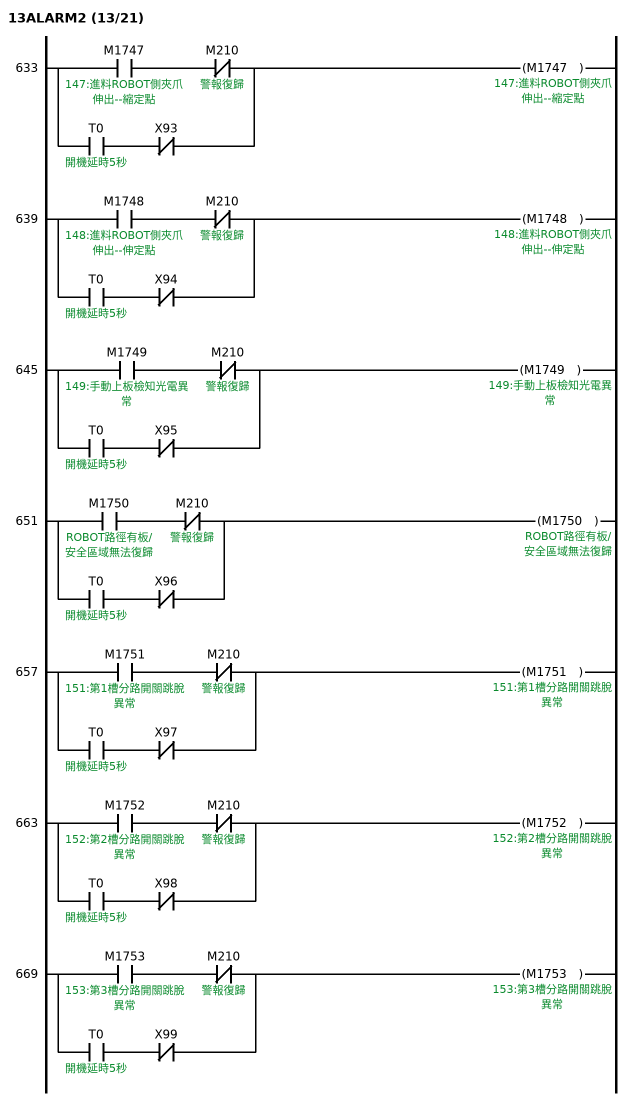
[picture p72: ladder of 13ALARM2, rungs at steps 633 to 669]
633   LD      M1747  ; 147:進料ROBOT側夾爪伸出--縮定點
      ANI     M210  ; 警報復歸
      LD      T0  ; 開機延時5秒
      ANI     X93
      ORB
      OUT     M1747  ; 147:進料ROBOT側夾爪伸出--縮定點
639   LD      M1748  ; 148:進料ROBOT側夾爪伸出--伸定點
      ANI     M210  ; 警報復歸
      LD      T0  ; 開機延時5秒
      ANI     X94
      ORB
      OUT     M1748  ; 148:進料ROBOT側夾爪伸出--伸定點
645   LD      M1749  ; 149:手動上板檢知光電異常
      ANI     M210  ; 警報復歸
      LD      T0  ; 開機延時5秒
      ANI     X95
      ORB
      OUT     M1749  ; 149:手動上板檢知光電異常
651   LD      M1750  ; ROBOT路徑有板/安全區域無法復歸
      ANI     M210  ; 警報復歸
      LD      T0  ; 開機延時5秒
      ANI     X96
      ORB
      OUT     M1750  ; ROBOT路徑有板/安全區域無法復歸
657   LD      M1751  ; 151:第1槽分路開關跳脫異常
      ANI     M210  ; 警報復歸
      LD      T0  ; 開機延時5秒
      ANI     X97
      ORB
      OUT     M1751  ; 151:第1槽分路開關跳脫異常
663   LD      M1752  ; 152:第2槽分路開關跳脫異常
      ANI     M210  ; 警報復歸
      LD      T0  ; 開機延時5秒
      ANI     X98
      ORB
      OUT     M1752  ; 152:第2槽分路開關跳脫異常
669   LD      M1753  ; 153:第3槽分路開關跳脫異常
      ANI     M210  ; 警報復歸
      LD      T0  ; 開機延時5秒
      ANI     X99
      ORB
      OUT     M1753  ; 153:第3槽分路開關跳脫異常
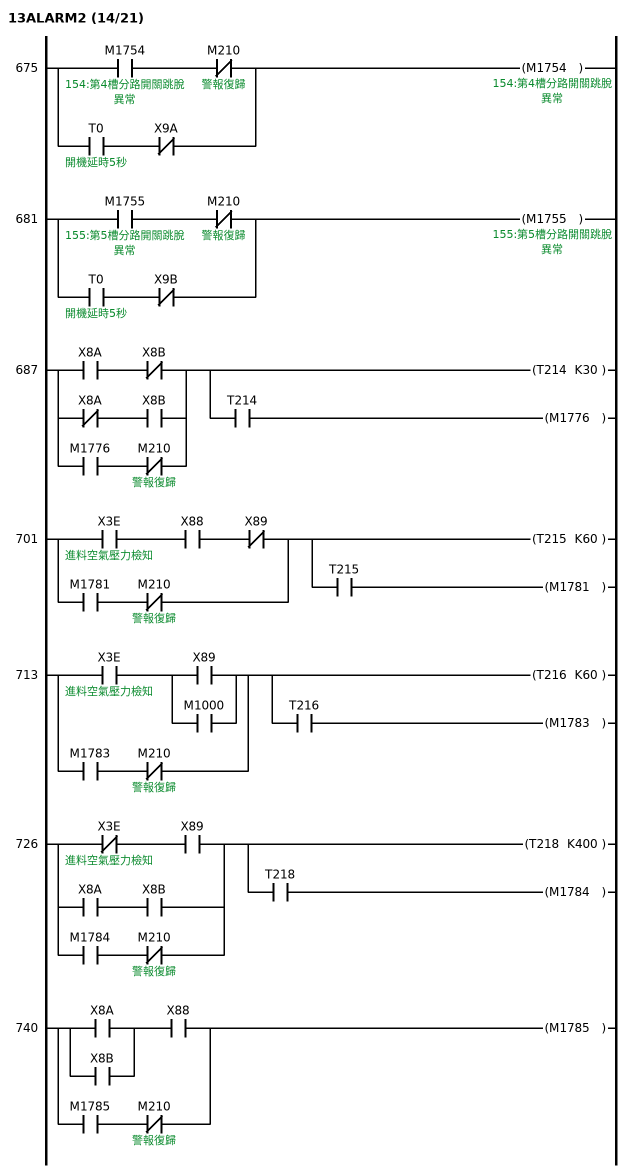
675   LD      M1754  ; 154:第4槽分路開關跳脫異常
      ANI     M210  ; 警報復歸
      LD      T0  ; 開機延時5秒
      ANI     X9A
      ORB
      OUT     M1754  ; 154:第4槽分路開關跳脫異常
681   LD      M1755  ; 155:第5槽分路開關跳脫異常
      ANI     M210  ; 警報復歸
      LD      T0  ; 開機延時5秒
      ANI     X9B
      ORB
      OUT     M1755  ; 155:第5槽分路開關跳脫異常
687   LD      X8A
      ANI     X8B
      LDI     X8A
      AND     X8B
      ORB
      LD      M1776
      ANI     M210  ; 警報復歸
      ORB
      OUT     T214 K30
      AND     T214
      OUT     M1776
701   LD      X3E  ; 進料空氣壓力檢知
      AND     X88
      ANI     X89
      LD      M1781
      ANI     M210  ; 警報復歸
      ORB
      OUT     T215 K60
      AND     T215
      OUT     M1781
713   LD      X3E  ; 進料空氣壓力檢知
      LD      X89
      OR      M1000
      ANB
      LD      M1783
      ANI     M210  ; 警報復歸
      ORB
      OUT     T216 K60
      AND     T216
      OUT     M1783
726   LDI     X3E  ; 進料空氣壓力檢知
      AND     X89
      LD      X8A
      AND     X8B
      ORB
      LD      M1784
      ANI     M210  ; 警報復歸
      ORB
      OUT     T218 K400
      AND     T218
      OUT     M1784
740   LD      X8A
      OR      X8B
      AND     X88
      LD      M1785
      ANI     M210  ; 警報復歸
      ORB
      OUT     M1785
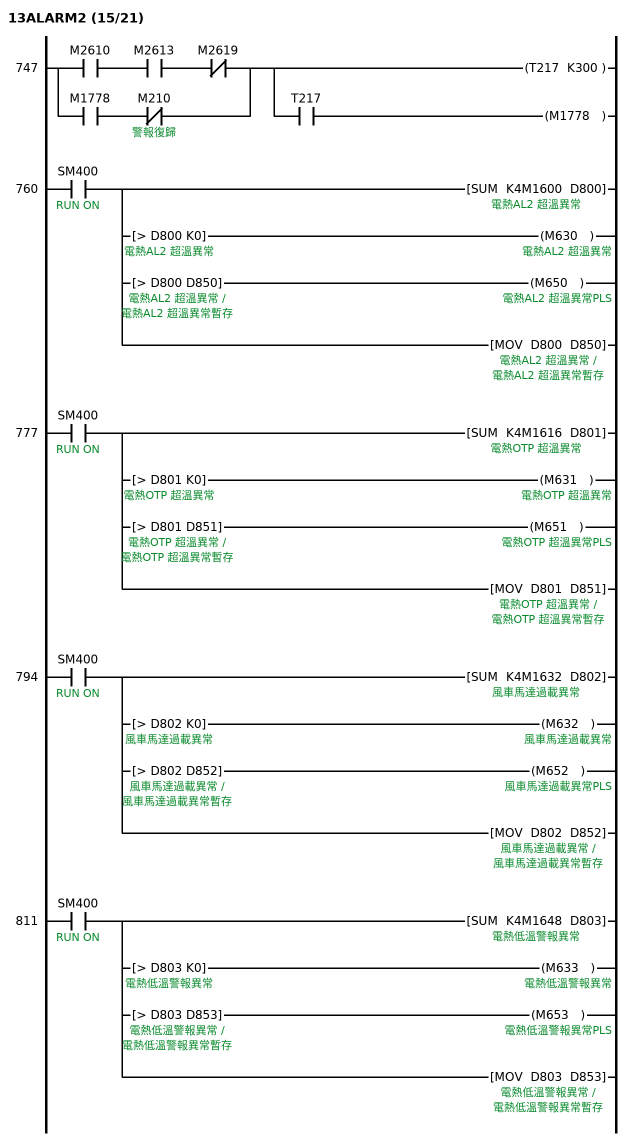
747   LD      M2610
      AND     M2613
      ANI     M2619
      LD      M1778
      ANI     M210  ; 警報復歸
      ORB
      OUT     T217 K300
      AND     T217
      OUT     M1778
760   LD      SM400  ; RUN ON
      SUM     K4M1600 D800  ; #01 電熱AL2 超溫 / 電熱AL2 超溫異常
      MPS
      AND>    D800 K0  ; 電熱AL2 超溫異常
      OUT     M630  ; 電熱AL2 超溫異常
      MRD
      AND>    D800 D850  ; 電熱AL2 超溫異常 / 電熱AL2 超溫異常暫存
      OUT     M650  ; 電熱AL2 超溫異常PLS
      MPP
      MOV     D800 D850
777   LD      SM400  ; RUN ON
      SUM     K4M1616 D801  ; #01 電熱OTP 超溫 / 電熱OTP 超溫異常
      MPS
      AND>    D801 K0  ; 電熱OTP 超溫異常
      OUT     M631  ; 電熱OTP 超溫異常
      MRD
      AND>    D801 D851  ; 電熱OTP 超溫異常 / 電熱OTP 超溫異常暫存
      OUT     M651  ; 電熱OTP 超溫異常PLS
      MPP
      MOV     D801 D851
794   LD      SM400  ; RUN ON
      SUM     K4M1632 D802  ; #01 風車過載 / 風車馬達過載異常
      MPS
      AND>    D802 K0  ; 風車馬達過載異常
      OUT     M632  ; 風車馬達過載異常
      MRD
      AND>    D802 D852  ; 風車馬達過載異常 / 風車馬達過載異常暫存
      OUT     M652  ; 風車馬達過載異常PLS
      MPP
      MOV     D802 D852
811   LD      SM400  ; RUN ON
      SUM     K4M1648 D803  ; #01 低溫警報 / 電熱低溫警報異常
      MPS
      AND>    D803 K0  ; 電熱低溫警報異常
      OUT     M633  ; 電熱低溫警報異常
      MRD
      AND>    D803 D853  ; 電熱低溫警報異常 / 電熱低溫警報異常暫存
      OUT     M653  ; 電熱低溫警報異常PLS
      MPP
      MOV     D803 D853
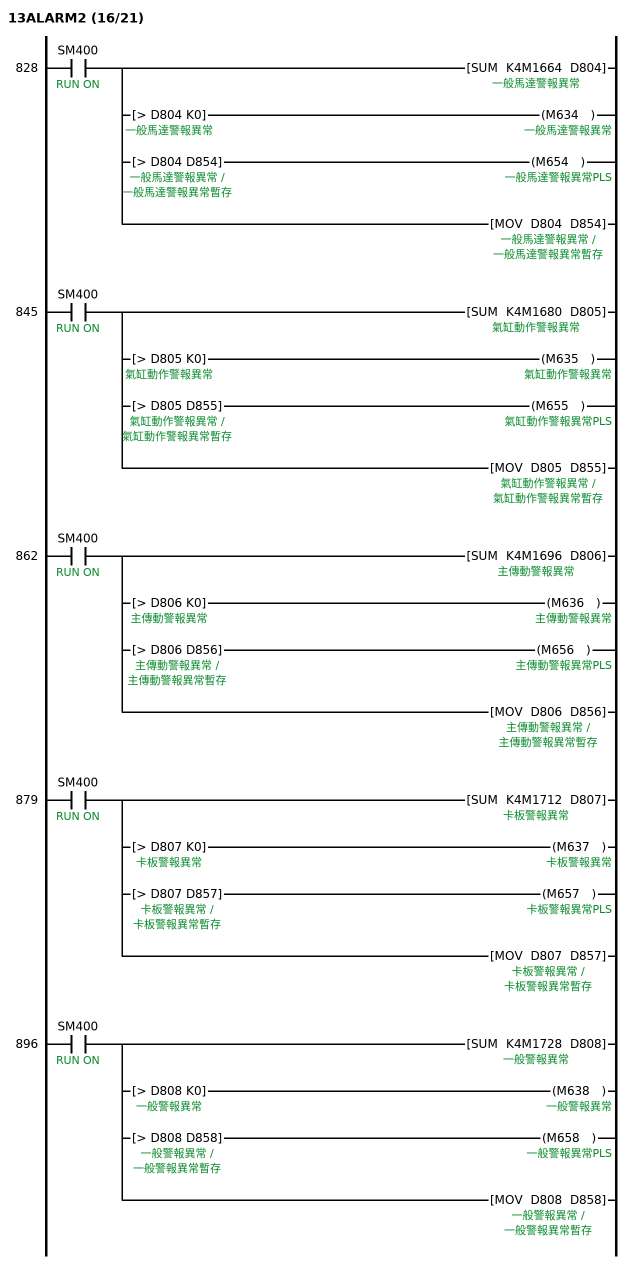
828   LD      SM400  ; RUN ON
      SUM     K4M1664 D804  ; 一般馬達警報異常
      MPS
      AND>    D804 K0  ; 一般馬達警報異常
      OUT     M634  ; 一般馬達警報異常
      MRD
      AND>    D804 D854  ; 一般馬達警報異常 / 一般馬達警報異常暫存
      OUT     M654  ; 一般馬達警報異常PLS
      MPP
      MOV     D804 D854
845   LD      SM400  ; RUN ON
      SUM     K4M1680 D805  ; 氣缸動作警報異常
      MPS
      AND>    D805 K0  ; 氣缸動作警報異常
      OUT     M635  ; 氣缸動作警報異常
      MRD
      AND>    D805 D855  ; 氣缸動作警報異常 / 氣缸動作警報異常暫存
      OUT     M655  ; 氣缸動作警報異常PLS
      MPP
      MOV     D805 D855
862   LD      SM400  ; RUN ON
      SUM     K4M1696 D806  ; 主傳動警報異常
      MPS
      AND>    D806 K0  ; 主傳動警報異常
      OUT     M636  ; 主傳動警報異常
      MRD
      AND>    D806 D856  ; 主傳動警報異常 / 主傳動警報異常暫存
      OUT     M656  ; 主傳動警報異常PLS
      MPP
      MOV     D806 D856
879   LD      SM400  ; RUN ON
      SUM     K4M1712 D807  ; 卡板警報異常
      MPS
      AND>    D807 K0  ; 卡板警報異常
      OUT     M637  ; 卡板警報異常
      MRD
      AND>    D807 D857  ; 卡板警報異常 / 卡板警報異常暫存
      OUT     M657  ; 卡板警報異常PLS
      MPP
      MOV     D807 D857
896   LD      SM400  ; RUN ON
      SUM     K4M1728 D808  ; 一般警報異常
      MPS
      AND>    D808 K0  ; 一般警報異常
      OUT     M638  ; 一般警報異常
      MRD
      AND>    D808 D858  ; 一般警報異常 / 一般警報異常暫存
      OUT     M658  ; 一般警報異常PLS
      MPP
      MOV     D808 D858
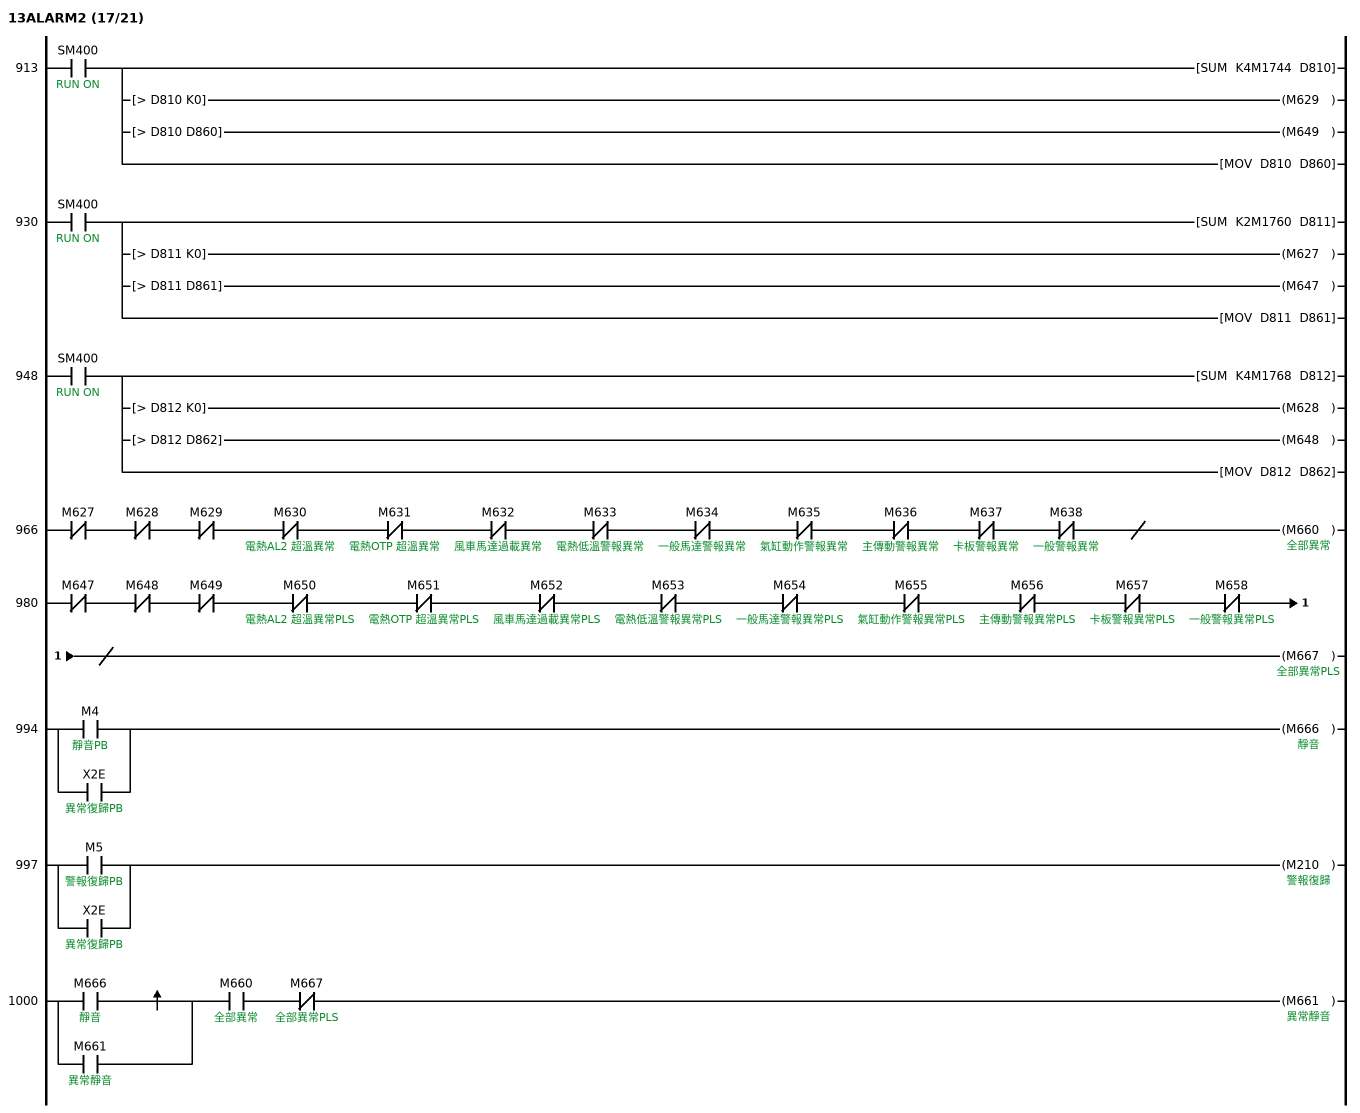
913   LD      SM400  ; RUN ON
      SUM     K4M1744 D810
      MPS
      AND>    D810 K0
      OUT     M629
      MRD
      AND>    D810 D860
      OUT     M649
      MPP
      MOV     D810 D860
930   LD      SM400  ; RUN ON
      SUM     K2M1760 D811
      MPS
      AND>    D811 K0
      OUT     M627
      MRD
      AND>    D811 D861
      OUT     M647
      MPP
      MOV     D811 D861
948   LD      SM400  ; RUN ON
      SUM     K4M1768 D812
      MPS
      AND>    D812 K0
      OUT     M628
      MRD
      AND>    D812 D862
      OUT     M648
      MPP
      MOV     D812 D862
966   LDI     M627
      ANI     M628
      ANI     M629
      ANI     M630  ; 電熱AL2 超溫異常
      ANI     M631  ; 電熱OTP 超溫異常
      ANI     M632  ; 風車馬達過載異常
      ANI     M633  ; 電熱低溫警報異常
      ANI     M634  ; 一般馬達警報異常
      ANI     M635  ; 氣缸動作警報異常
      ANI     M636  ; 主傳動警報異常
      ANI     M637  ; 卡板警報異常
      ANI     M638  ; 一般警報異常
      INV
      OUT     M660  ; 全部異常
980   LDI     M647
      ANI     M648
      ANI     M649
      ANI     M650  ; 電熱AL2 超溫異常PLS
      ANI     M651  ; 電熱OTP 超溫異常PLS
      ANI     M652  ; 風車馬達過載異常PLS
      ANI     M653  ; 電熱低溫警報異常PLS
      ANI     M654  ; 一般馬達警報異常PLS
      ANI     M655  ; 氣缸動作警報異常PLS
      ANI     M656  ; 主傳動警報異常PLS
      ANI     M657  ; 卡板警報異常PLS
      ANI     M658  ; 一般警報異常PLS
      INV
      OUT     M667  ; 全部異常PLS
994   LD      M4  ; 靜音PB
      OR      X2E  ; 異常復歸PB
      OUT     M666  ; 靜音
997   LD      M5  ; 警報復歸PB
      OR      X2E  ; 異常復歸PB
      OUT     M210  ; 警報復歸
1000  LD      M666  ; 靜音
      MEP
      OR      M661  ; 異常靜音
      AND     M660  ; 全部異常
      ANI     M667  ; 全部異常PLS
      OUT     M661  ; 異常靜音
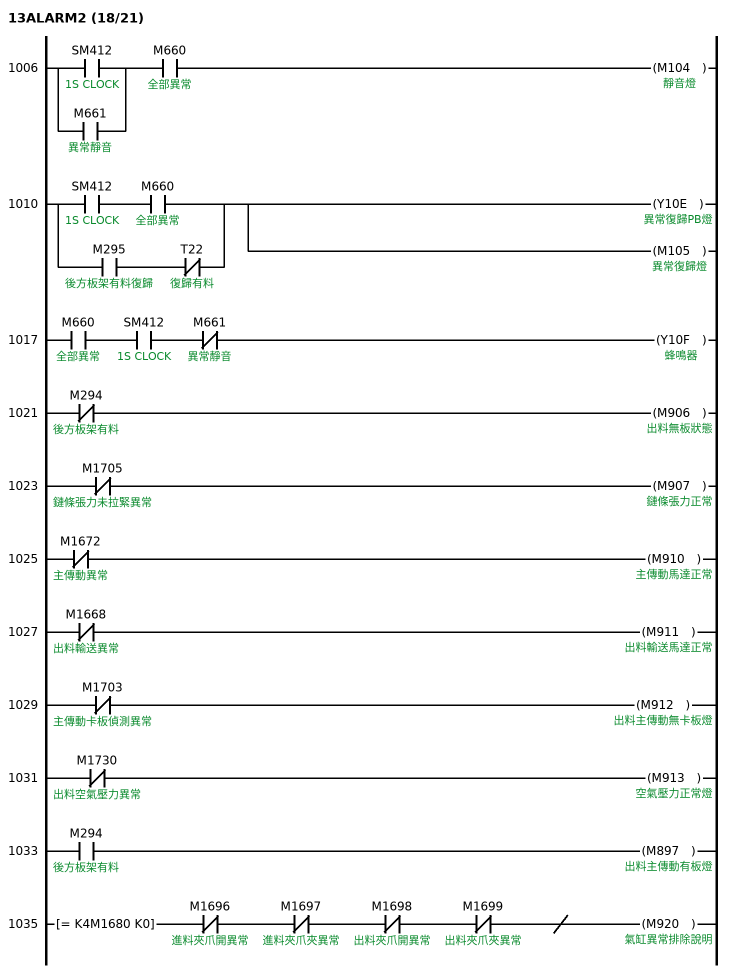
1006  LD      SM412  ; 1S CLOCK
      OR      M661  ; 異常靜音
      AND     M660  ; 全部異常
      OUT     M104  ; 靜音燈
1010  LD      SM412  ; 1S CLOCK
      AND     M660  ; 全部異常
      LD      M295  ; 後方板架有料復歸
      ANI     T22  ; 復歸有料
      ORB
      OUT     Y10E  ; 異常復歸PB燈
      OUT     M105  ; 異常復歸燈
1017  LD      M660  ; 全部異常
      AND     SM412  ; 1S CLOCK
      ANI     M661  ; 異常靜音
      OUT     Y10F  ; 蜂鳴器
1021  LDI     M294  ; 後方板架有料
      OUT     M906  ; 出料無板狀態
1023  LDI     M1705  ; 鏈條張力未拉緊異常
      OUT     M907  ; 鏈條張力正常
1025  LDI     M1672  ; 主傳動異常
      OUT     M910  ; 主傳動馬達正常
1027  LDI     M1668  ; 出料輸送異常
      OUT     M911  ; 出料輸送馬達正常
1029  LDI     M1703  ; 主傳動卡板偵測異常
      OUT     M912  ; 出料主傳動無卡板燈
1031  LDI     M1730  ; 出料空氣壓力異常
      OUT     M913  ; 空氣壓力正常燈
1033  LD      M294  ; 後方板架有料
      OUT     M897  ; 出料主傳動有板燈
1035  LD=     K4M1680 K0  ; 上料手臂前夾爪放異常
      ANI     M1696  ; 進料夾爪開異常
      ANI     M1697  ; 進料夾爪夾異常
      ANI     M1698  ; 出料夾爪開異常
      ANI     M1699  ; 出料夾爪夾異常
      INV
      OUT     M920  ; 氣缸異常排除說明
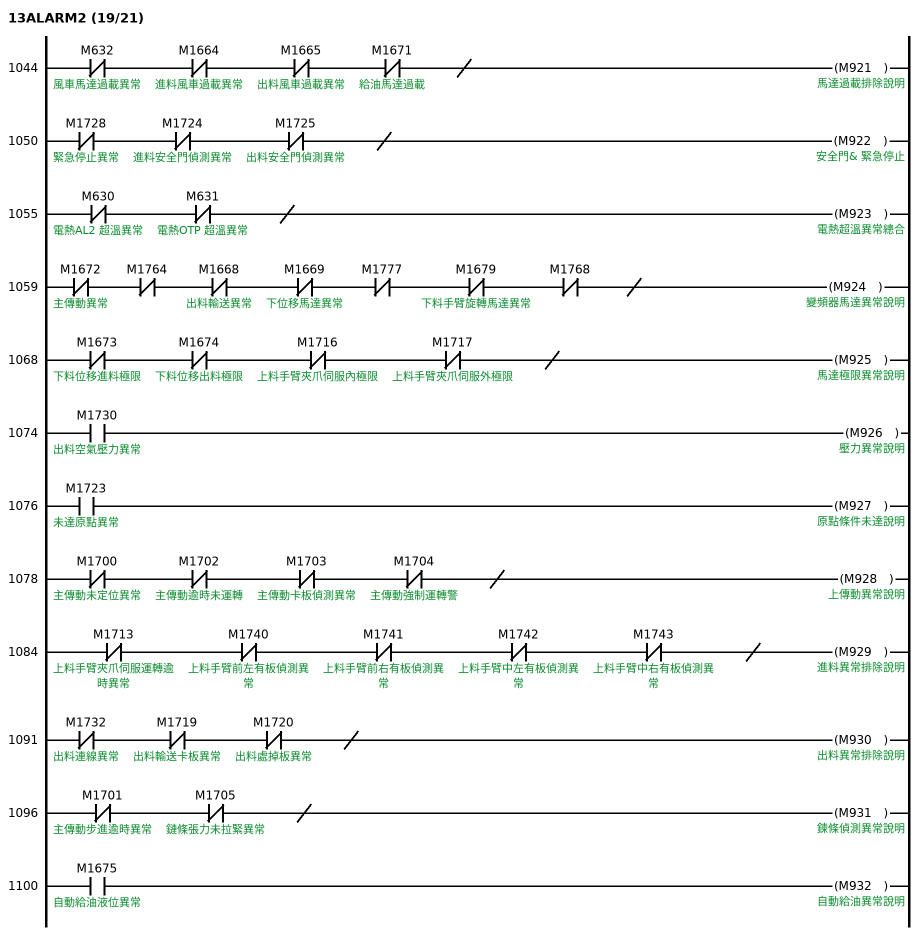
1044  LDI     M632  ; 風車馬達過載異常
      ANI     M1664  ; 進料風車過載異常
      ANI     M1665  ; 出料風車過載異常
      ANI     M1671  ; 給油馬達過載
      INV
      OUT     M921  ; 馬達過載排除說明
1050  LDI     M1728  ; 緊急停止異常
      ANI     M1724  ; 進料安全門偵測異常
      ANI     M1725  ; 出料安全門偵測異常
      INV
      OUT     M922  ; 安全門& 緊急停止
1055  LDI     M630  ; 電熱AL2 超溫異常
      ANI     M631  ; 電熱OTP 超溫異常
      INV
      OUT     M923  ; 電熱超溫異常總合
1059  LDI     M1672  ; 主傳動異常
      ANI     M1764
      ANI     M1668  ; 出料輸送異常
      ANI     M1669  ; 下位移馬達異常
      ANI     M1777
      ANI     M1679  ; 下料手臂旋轉馬達異常
      ANI     M1768
      INV
      OUT     M924  ; 變頻器馬達異常說明
1068  LDI     M1673  ; 下料位移進料極限
      ANI     M1674  ; 下料位移出料極限
      ANI     M1716  ; 上料手臂夾爪伺服內極限
      ANI     M1717  ; 上料手臂夾爪伺服外極限
      INV
      OUT     M925  ; 馬達極限異常說明
1074  LD      M1730  ; 出料空氣壓力異常
      OUT     M926  ; 壓力異常說明
1076  LD      M1723  ; 未達原點異常
      OUT     M927  ; 原點條件未達說明
1078  LDI     M1700  ; 主傳動未定位異常
      ANI     M1702  ; 主傳動逾時未運轉
      ANI     M1703  ; 主傳動卡板偵測異常
      ANI     M1704  ; 主傳動強制運轉警
      INV
      OUT     M928  ; 上傳動異常說明
1084  LDI     M1713  ; 上料手臂夾爪伺服運轉逾時異常
      ANI     M1740  ; 上料手臂前左有板偵測異常
      ANI     M1741  ; 上料手臂前右有板偵測異常
      ANI     M1742  ; 上料手臂中左有板偵測異常
      ANI     M1743  ; 上料手臂中右有板偵測異常
      INV
      OUT     M929  ; 進料異常排除說明
1091  LDI     M1732  ; 出料連線異常
      ANI     M1719  ; 出料輸送卡板異常
      ANI     M1720  ; 出料處掉板異常
      INV
      OUT     M930  ; 出料異常排除說明
1096  LDI     M1701  ; 主傳動步進逾時異常
      ANI     M1705  ; 鏈條張力未拉緊異常
      INV
      OUT     M931  ; 鍊條偵測異常說明
1100  LD      M1675  ; 自動給油液位異常
      OUT     M932  ; 自動給油異常說明
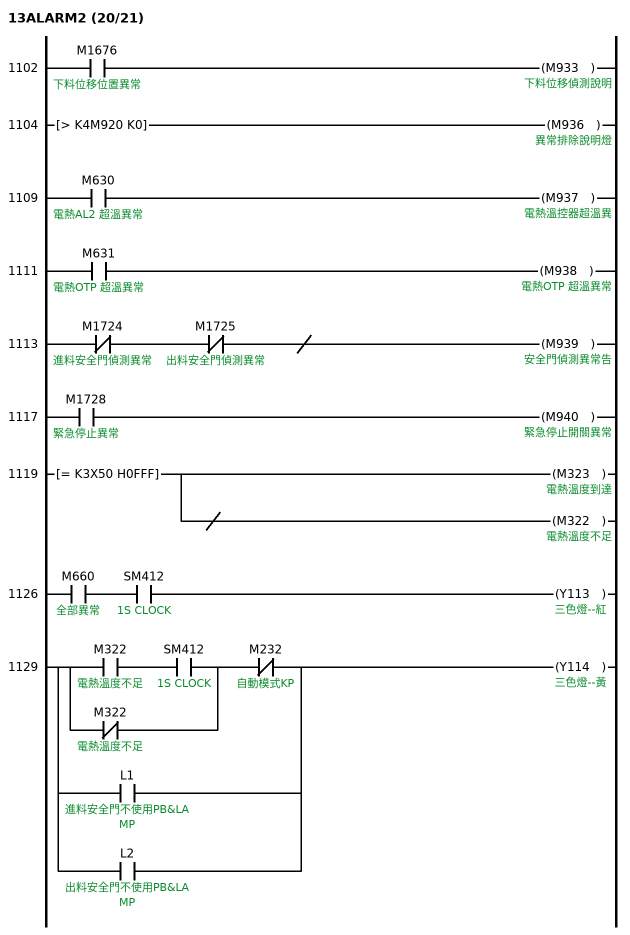
1102  LD      M1676  ; 下料位移位置異常
      OUT     M933  ; 下料位移偵測說明
1104  LD>     K4M920 K0  ; 氣缸異常排除說明
      OUT     M936  ; 異常排除說明燈
1109  LD      M630  ; 電熱AL2 超溫異常
      OUT     M937  ; 電熱溫控器超溫異
1111  LD      M631  ; 電熱OTP 超溫異常
      OUT     M938  ; 電熱OTP 超溫異常
1113  LDI     M1724  ; 進料安全門偵測異常
      ANI     M1725  ; 出料安全門偵測異常
      INV
      OUT     M939  ; 安全門偵測異常告
1117  LD      M1728  ; 緊急停止異常
      OUT     M940  ; 緊急停止開關異常
1119  LD=     K3X50 H0FFF  ; #01 溫度到達AL1
      OUT     M323  ; 電熱溫度到達
      INV
      OUT     M322  ; 電熱溫度不足
1126  LD      M660  ; 全部異常
      AND     SM412  ; 1S CLOCK
      OUT     Y113  ; 三色燈--紅
1129  LD      M322  ; 電熱溫度不足
      AND     SM412  ; 1S CLOCK
      ORI     M322  ; 電熱溫度不足
      ANI     M232  ; 自動模式KP
      OR      L1  ; 進料安全門不使用PB&LAMP
      OR      L2  ; 出料安全門不使用PB&LAMP
      OUT     Y114  ; 三色燈--黃
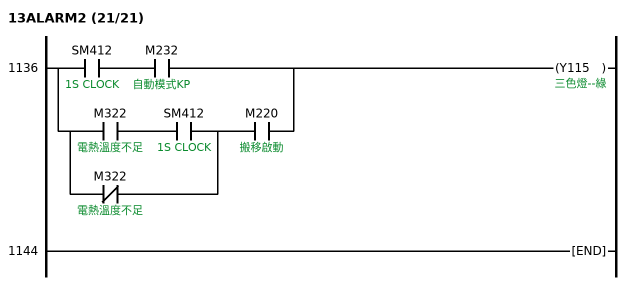
1136  LD      SM412  ; 1S CLOCK
      AND     M232  ; 自動模式KP
      LD      M322  ; 電熱溫度不足
      AND     SM412  ; 1S CLOCK
      ORI     M322  ; 電熱溫度不足
      AND     M220  ; 搬移啟動
      ORB
      OUT     Y115  ; 三色燈--綠
1144  END
END_PROGRAM

PROGRAM 14TIME
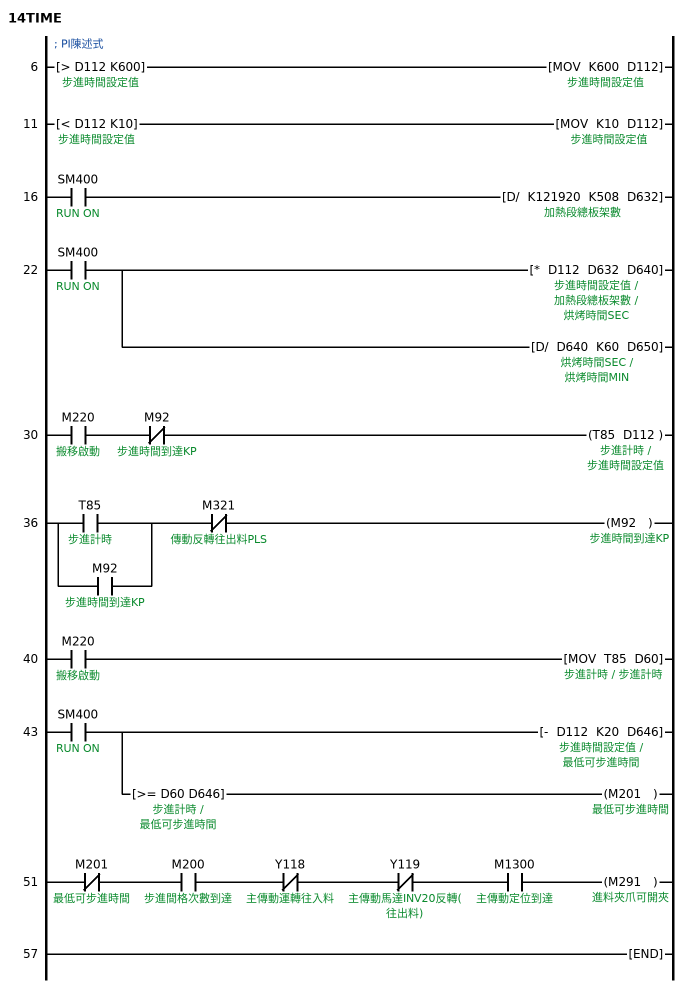
; PI陳述式
6     LD>     D112 K600  ; 步進時間設定值
      MOV     K600 D112
11    LD<     D112 K10  ; 步進時間設定值
      MOV     K10 D112
16    LD      SM400  ; RUN ON
      D/      K121920 K508 D632  ; 加熱段總板架數
22    LD      SM400  ; RUN ON
      *       D112 D632 D640  ; 烘烤時間SEC
      D/      D640 K60 D650  ; 烘烤時間MIN
30    LD      M220  ; 搬移啟動
      ANI     M92  ; 步進時間到達KP
      OUT     T85 D112  ; 步進計時 / 步進時間設定值
36    LD      T85  ; 步進計時
      OR      M92  ; 步進時間到達KP
      ANI     M321  ; 傳動反轉往出料PLS
      OUT     M92  ; 步進時間到達KP
40    LD      M220  ; 搬移啟動
      MOV     T85 D60  ; 步進計時
43    LD      SM400  ; RUN ON
      -       D112 K20 D646  ; 最低可步進時間
      AND>=   D60 D646  ; 步進計時 / 最低可步進時間
      OUT     M201  ; 最低可步進時間
51    LDI     M201  ; 最低可步進時間
      AND     M200  ; 步進間格次數到達
      ANI     Y118  ; 主傳動運轉往入料
      ANI     Y119  ; 主傳動馬達INV20反轉(往出料)
      AND     M1300  ; 主傳動定位到達
      OUT     M291  ; 進料夾爪可開夾
57    END
END_PROGRAM

PROGRAM 15STATUS
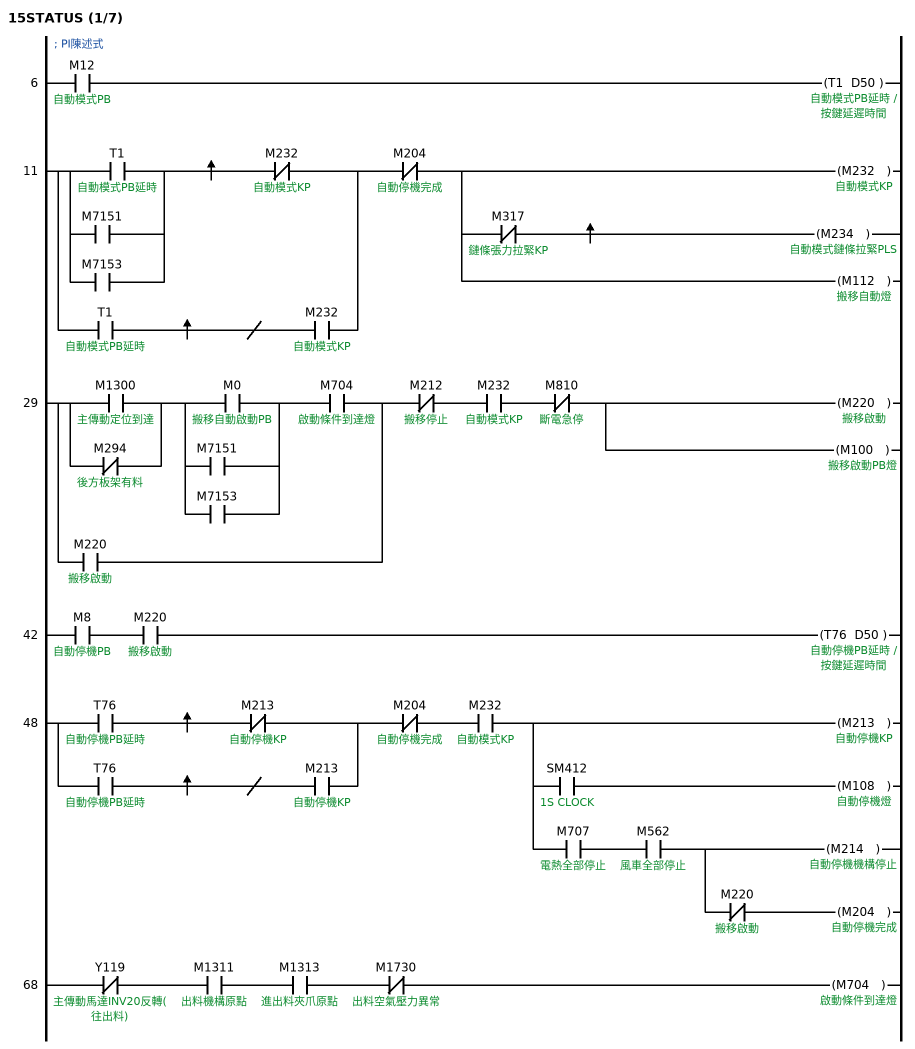
; PI陳述式
6     LD      M12  ; 自動模式PB
      OUT     T1 D50  ; 自動模式PB延時 / 按鍵延遲時間
11    LD      T1  ; 自動模式PB延時
      OR      M7151
      OR      M7153
      MEP
      ANI     M232  ; 自動模式KP
      LD      T1  ; 自動模式PB延時
      MEP
      INV
      AND     M232  ; 自動模式KP
      ORB
      ANI     M204  ; 自動停機完成
      OUT     M232  ; 自動模式KP
      MPS
      ANI     M317  ; 鏈條張力拉緊KP
      MEP
      OUT     M234  ; 自動模式鏈條拉緊PLS
      MPP
      OUT     M112  ; 搬移自動燈
29    LD      M1300  ; 主傳動定位到達
      ORI     M294  ; 後方板架有料
      LD      M0  ; 搬移自動啟動PB
      OR      M7151
      OR      M7153
      ANB
      AND     M704  ; 啟動條件到達燈
      OR      M220  ; 搬移啟動
      ANI     M212  ; 搬移停止
      AND     M232  ; 自動模式KP
      ANI     M810  ; 斷電急停
      OUT     M220  ; 搬移啟動
      OUT     M100  ; 搬移啟動PB燈
42    LD      M8  ; 自動停機PB
      AND     M220  ; 搬移啟動
      OUT     T76 D50  ; 自動停機PB延時 / 按鍵延遲時間
48    LD      T76  ; 自動停機PB延時
      MEP
      ANI     M213  ; 自動停機KP
      LD      T76  ; 自動停機PB延時
      MEP
      INV
      AND     M213  ; 自動停機KP
      ORB
      ANI     M204  ; 自動停機完成
      AND     M232  ; 自動模式KP
      OUT     M213  ; 自動停機KP
      MPS
      AND     SM412  ; 1S CLOCK
      OUT     M108  ; 自動停機燈
      MPP
      AND     M707  ; 電熱全部停止
      AND     M562  ; 風車全部停止
      OUT     M214  ; 自動停機機構停止
      ANI     M220  ; 搬移啟動
      OUT     M204  ; 自動停機完成
68    LDI     Y119  ; 主傳動馬達INV20反轉(往出料)
      AND     M1311  ; 出料機構原點
      AND     M1313  ; 進出料夾爪原點
      ANI     M1730  ; 出料空氣壓力異常
      OUT     M704  ; 啟動條件到達燈
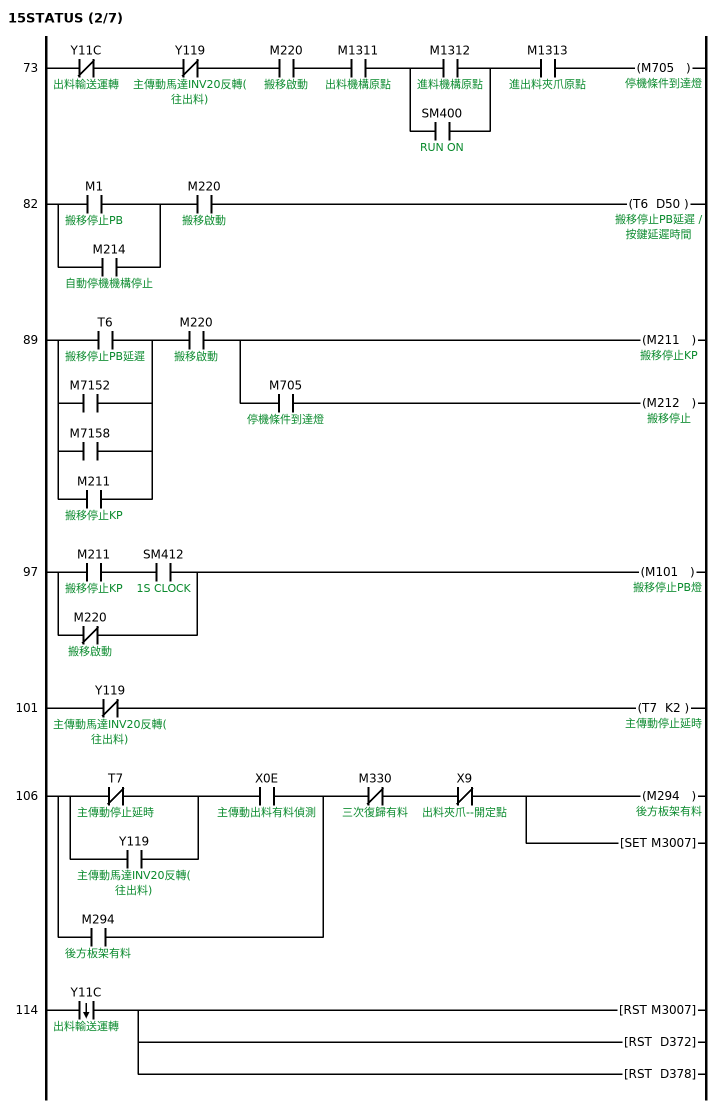
73    LDI     Y11C  ; 出料輸送運轉
      ANI     Y119  ; 主傳動馬達INV20反轉(往出料)
      AND     M220  ; 搬移啟動
      AND     M1311  ; 出料機構原點
      LD      M1312  ; 進料機構原點
      OR      SM400  ; RUN ON
      ANB
      AND     M1313  ; 進出料夾爪原點
      OUT     M705  ; 停機條件到達燈
82    LD      M1  ; 搬移停止PB
      OR      M214  ; 自動停機機構停止
      AND     M220  ; 搬移啟動
      OUT     T6 D50  ; 搬移停止PB延遲 / 按鍵延遲時間
89    LD      T6  ; 搬移停止PB延遲
      OR      M7152
      OR      M7158
      OR      M211  ; 搬移停止KP
      AND     M220  ; 搬移啟動
      OUT     M211  ; 搬移停止KP
      AND     M705  ; 停機條件到達燈
      OUT     M212  ; 搬移停止
97    LD      M211  ; 搬移停止KP
      AND     SM412  ; 1S CLOCK
      ORI     M220  ; 搬移啟動
      OUT     M101  ; 搬移停止PB燈
101   LDI     Y119  ; 主傳動馬達INV20反轉(往出料)
      OUT     T7 K2  ; 主傳動停止延時
106   LDI     T7  ; 主傳動停止延時
      OR      Y119  ; 主傳動馬達INV20反轉(往出料)
      AND     X0E  ; 主傳動出料有料偵測
      OR      M294  ; 後方板架有料
      ANI     M330  ; 三次復歸有料
      ANI     X9  ; 出料夾爪--開定點
      OUT     M294  ; 後方板架有料
      SET     M3007
114   LDF     Y11C  ; 出料輸送運轉
      RST     M3007
      RST     D372
      RST     D378
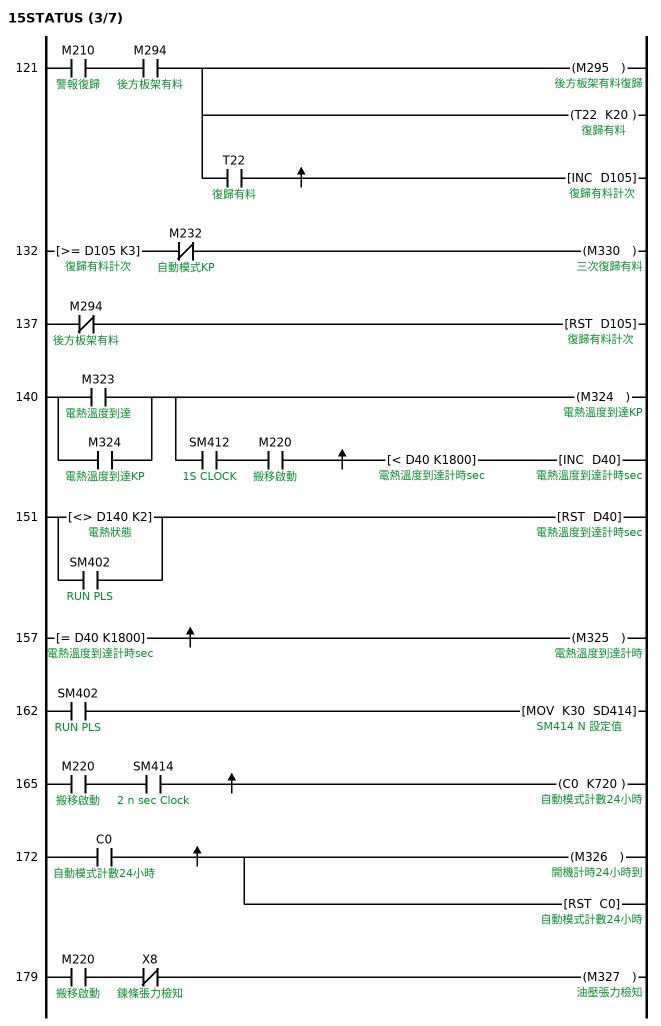
121   LD      M210  ; 警報復歸
      AND     M294  ; 後方板架有料
      OUT     M295  ; 後方板架有料復歸
      OUT     T22 K20  ; 復歸有料
      AND     T22  ; 復歸有料
      MEP
      INC     D105  ; 復歸有料計次
132   LD>=    D105 K3  ; 復歸有料計次
      ANI     M232  ; 自動模式KP
      OUT     M330  ; 三次復歸有料
137   LDI     M294  ; 後方板架有料
      RST     D105  ; 復歸有料計次
140   LD      M323  ; 電熱溫度到達
      OR      M324  ; 電熱溫度到達KP
      OUT     M324  ; 電熱溫度到達KP
      AND     SM412  ; 1S CLOCK
      AND     M220  ; 搬移啟動
      MEP
      AND<    D40 K1800  ; 電熱溫度到達計時sec
      INC     D40
151   LD<>    D140 K2  ; 電熱狀態
      OR      SM402  ; RUN PLS
      RST     D40  ; 電熱溫度到達計時sec
157   LD=     D40 K1800  ; 電熱溫度到達計時sec
      MEP
      OUT     M325  ; 電熱溫度到達計時
162   LD      SM402  ; RUN PLS
      MOV     K30 SD414  ; SM414 N 設定值
165   LD      M220  ; 搬移啟動
      AND     SM414  ; 2 n sec Clock
      MEP
      OUT     C0 K720  ; 自動模式計數24小時
172   LD      C0  ; 自動模式計數24小時
      MEP
      OUT     M326  ; 開機計時24小時到
      RST     C0  ; 自動模式計數24小時
179   LD      M220  ; 搬移啟動
      ANI     X8  ; 鍊條張力檢知
      OUT     M327  ; 油壓張力檢知
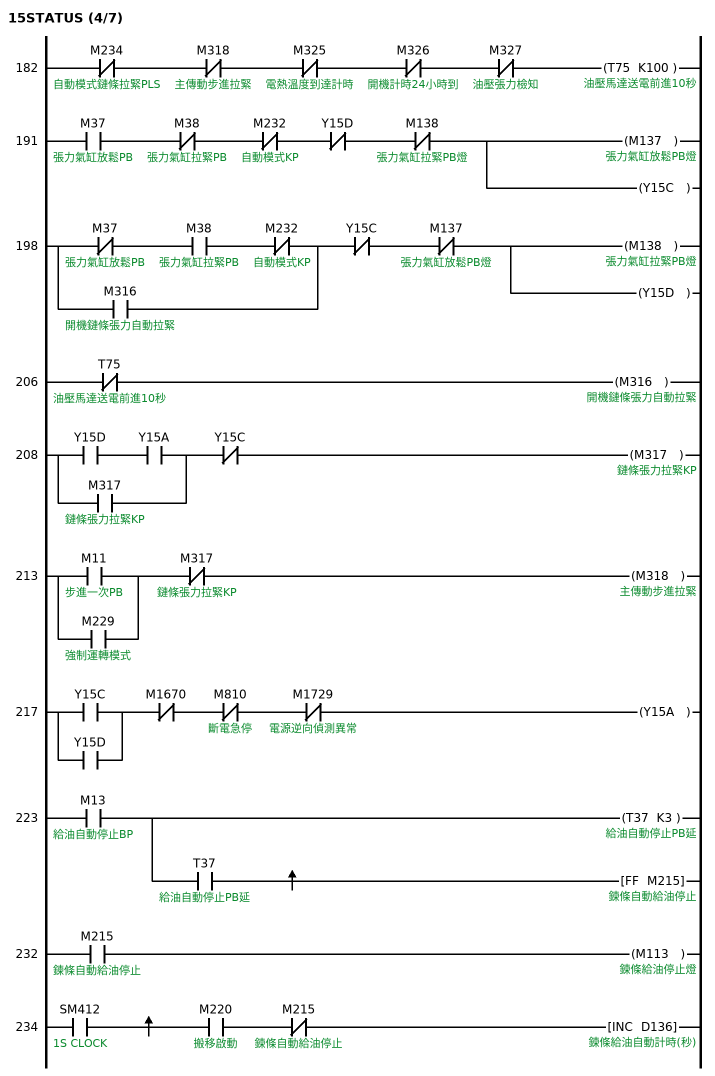
182   LDI     M234  ; 自動模式鏈條拉緊PLS
      ANI     M318  ; 主傳動步進拉緊
      ANI     M325  ; 電熱溫度到達計時
      ANI     M326  ; 開機計時24小時到
      ANI     M327  ; 油壓張力檢知
      OUT     T75 K100  ; 油壓馬達送電前進10秒
191   LD      M37  ; 張力氣缸放鬆PB
      ANI     M38  ; 張力氣缸拉緊PB
      ANI     M232  ; 自動模式KP
      ANI     Y15D
      ANI     M138  ; 張力氣缸拉緊PB燈
      OUT     M137  ; 張力氣缸放鬆PB燈
      OUT     Y15C
198   LDI     M37  ; 張力氣缸放鬆PB
      AND     M38  ; 張力氣缸拉緊PB
      ANI     M232  ; 自動模式KP
      OR      M316  ; 開機鏈條張力自動拉緊
      ANI     Y15C
      ANI     M137  ; 張力氣缸放鬆PB燈
      OUT     M138  ; 張力氣缸拉緊PB燈
      OUT     Y15D
206   LDI     T75  ; 油壓馬達送電前進10秒
      OUT     M316  ; 開機鏈條張力自動拉緊
208   LD      Y15D
      AND     Y15A
      OR      M317  ; 鏈條張力拉緊KP
      ANI     Y15C
      OUT     M317  ; 鏈條張力拉緊KP
213   LD      M11  ; 步進一次PB
      OR      M229  ; 強制運轉模式
      ANI     M317  ; 鏈條張力拉緊KP
      OUT     M318  ; 主傳動步進拉緊
217   LD      Y15C
      OR      Y15D
      ANI     M1670
      ANI     M810  ; 斷電急停
      ANI     M1729  ; 電源逆向偵測異常
      OUT     Y15A
223   LD      M13  ; 給油自動停止BP
      OUT     T37 K3  ; 給油自動停止PB延
      AND     T37  ; 給油自動停止PB延
      MEP
      FF      M215  ; 鍊條自動給油停止
232   LD      M215  ; 鍊條自動給油停止
      OUT     M113  ; 鍊條給油停止燈
234   LD      SM412  ; 1S CLOCK
      MEP
      AND     M220  ; 搬移啟動
      ANI     M215  ; 鍊條自動給油停止
      INC     D136  ; 鍊條給油自動計時(秒)
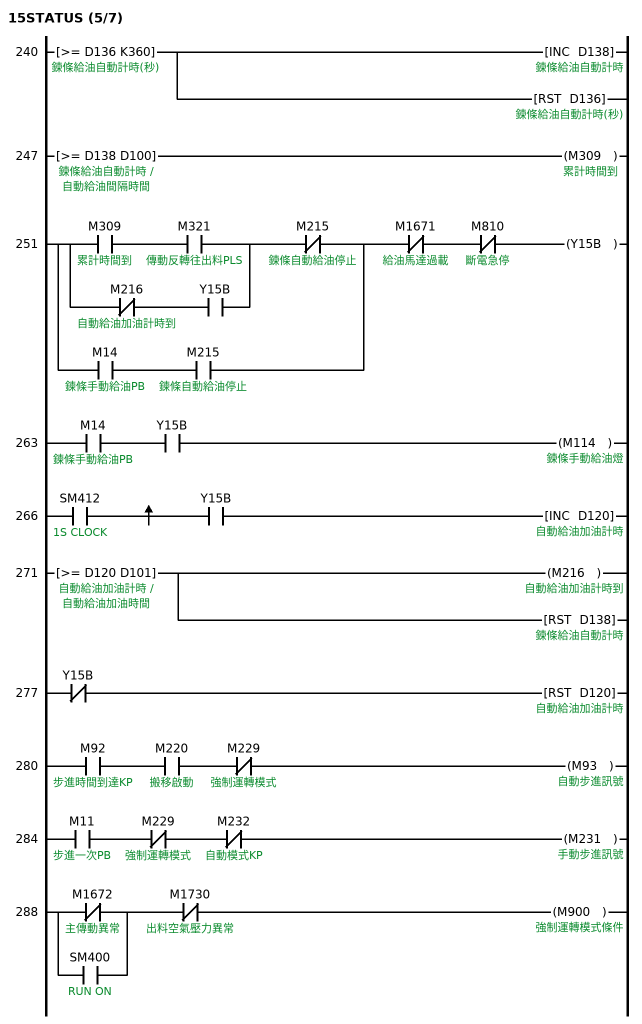
240   LD>=    D136 K360  ; 鍊條給油自動計時(秒)
      INC     D138  ; 鍊條給油自動計時
      RST     D136  ; 鍊條給油自動計時(秒)
247   LD>=    D138 D100  ; 鍊條給油自動計時 / 自動給油間隔時間
      OUT     M309  ; 累計時間到
251   LD      M309  ; 累計時間到
      AND     M321  ; 傳動反轉往出料PLS
      LDI     M216  ; 自動給油加油計時到
      AND     Y15B
      ORB
      ANI     M215  ; 鍊條自動給油停止
      LD      M14  ; 鍊條手動給油PB
      AND     M215  ; 鍊條自動給油停止
      ORB
      ANI     M1671  ; 給油馬達過載
      ANI     M810  ; 斷電急停
      OUT     Y15B
263   LD      M14  ; 鍊條手動給油PB
      AND     Y15B
      OUT     M114  ; 鍊條手動給油燈
266   LD      SM412  ; 1S CLOCK
      MEP
      AND     Y15B
      INC     D120  ; 自動給油加油計時
271   LD>=    D120 D101  ; 自動給油加油計時 / 自動給油加油時間
      OUT     M216  ; 自動給油加油計時到
      RST     D138  ; 鍊條給油自動計時
277   LDI     Y15B
      RST     D120  ; 自動給油加油計時
280   LD      M92  ; 步進時間到達KP
      AND     M220  ; 搬移啟動
      ANI     M229  ; 強制運轉模式
      OUT     M93  ; 自動步進訊號
284   LD      M11  ; 步進一次PB
      ANI     M229  ; 強制運轉模式
      ANI     M232  ; 自動模式KP
      OUT     M231  ; 手動步進訊號
288   LDI     M1672  ; 主傳動異常
      OR      SM400  ; RUN ON
      ANI     M1730  ; 出料空氣壓力異常
      OUT     M900  ; 強制運轉模式條件
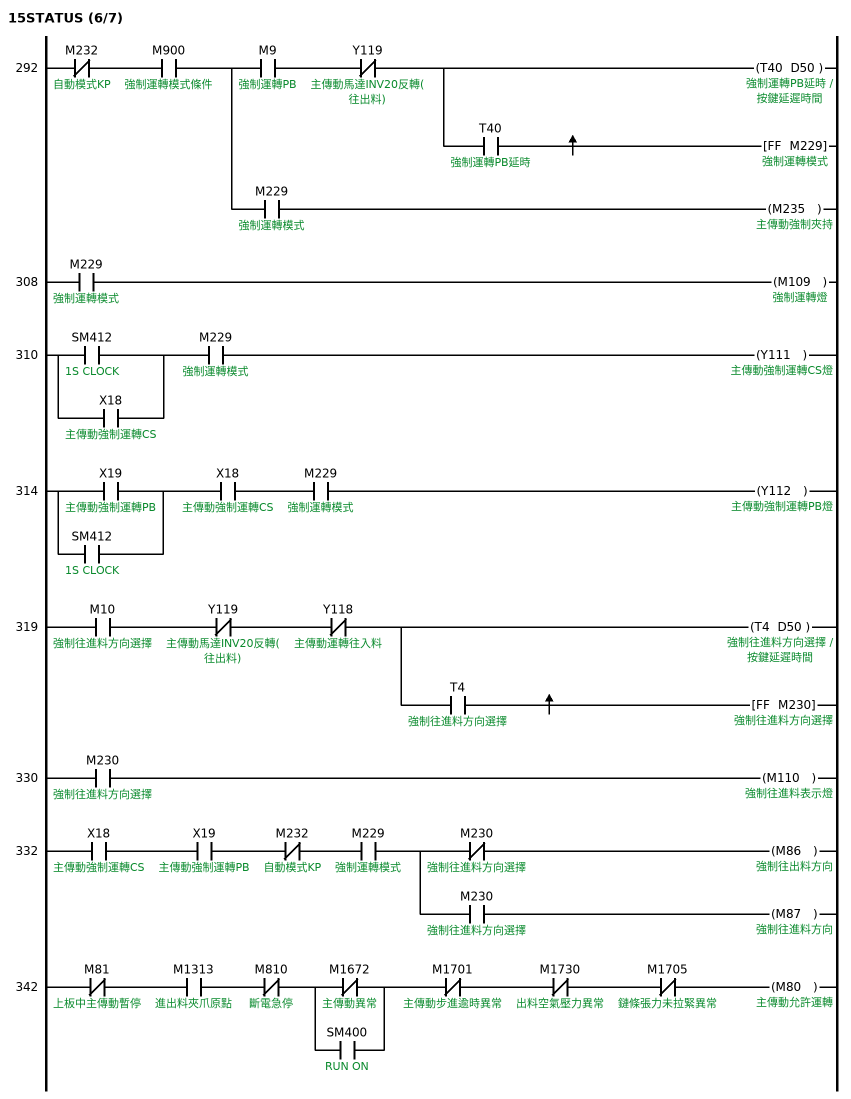
292   LDI     M232  ; 自動模式KP
      AND     M900  ; 強制運轉模式條件
      MPS
      AND     M9  ; 強制運轉PB
      ANI     Y119  ; 主傳動馬達INV20反轉(往出料)
      OUT     T40 D50  ; 強制運轉PB延時 / 按鍵延遲時間
      AND     T40  ; 強制運轉PB延時
      MEP
      FF      M229
      MPP
      AND     M229  ; 強制運轉模式
      OUT     M235  ; 主傳動強制夾持
308   LD      M229  ; 強制運轉模式
      OUT     M109  ; 強制運轉燈
310   LD      SM412  ; 1S CLOCK
      OR      X18  ; 主傳動強制運轉CS
      AND     M229  ; 強制運轉模式
      OUT     Y111  ; 主傳動強制運轉CS燈
314   LD      X19  ; 主傳動強制運轉PB
      OR      SM412  ; 1S CLOCK
      AND     X18  ; 主傳動強制運轉CS
      AND     M229  ; 強制運轉模式
      OUT     Y112  ; 主傳動強制運轉PB燈
319   LD      M10  ; 強制往進料方向選擇
      ANI     Y119  ; 主傳動馬達INV20反轉(往出料)
      ANI     Y118  ; 主傳動運轉往入料
      OUT     T4 D50  ; 強制往進料方向選擇 / 按鍵延遲時間
      AND     T4  ; 強制往進料方向選擇
      MEP
      FF      M230  ; 強制往進料方向選擇
330   LD      M230  ; 強制往進料方向選擇
      OUT     M110  ; 強制往進料表示燈
332   LD      X18  ; 主傳動強制運轉CS
      AND     X19  ; 主傳動強制運轉PB
      ANI     M232  ; 自動模式KP
      AND     M229  ; 強制運轉模式
      MPS
      ANI     M230  ; 強制往進料方向選擇
      OUT     M86  ; 強制往出料方向
      MPP
      AND     M230  ; 強制往進料方向選擇
      OUT     M87  ; 強制往進料方向
342   LDI     M81  ; 上板中主傳動暫停
      AND     M1313  ; 進出料夾爪原點
      ANI     M810  ; 斷電急停
      LDI     M1672  ; 主傳動異常
      OR      SM400  ; RUN ON
      ANB
      ANI     M1701  ; 主傳動步進逾時異常
      ANI     M1730  ; 出料空氣壓力異常
      ANI     M1705  ; 鏈條張力未拉緊異常
      OUT     M80  ; 主傳動允許運轉
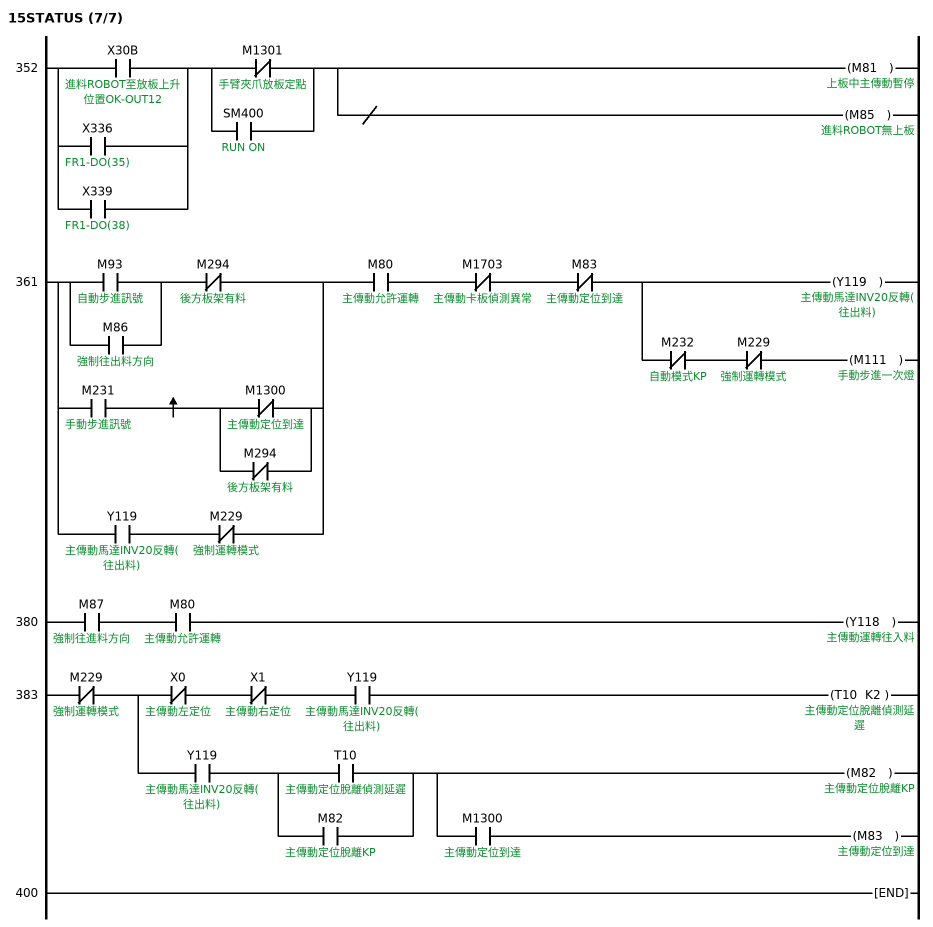
352   LD      X30B  ; 進料ROBOT至放板上升位置OK-OUT12
      OR      X336  ; FR1-DO(35)
      OR      X339  ; FR1-DO(38)
      LDI     M1301  ; 手臂夾爪放板定點
      OR      SM400  ; RUN ON
      ANB
      OUT     M81  ; 上板中主傳動暫停
      INV
      OUT     M85  ; 進料ROBOT無上板
361   LD      M93  ; 自動步進訊號
      OR      M86  ; 強制往出料方向
      ANI     M294  ; 後方板架有料
      LD      M231  ; 手動步進訊號
      MEP
      LDI     M1300  ; 主傳動定位到達
      ORI     M294  ; 後方板架有料
      ANB
      ORB
      LD      Y119  ; 主傳動馬達INV20反轉(往出料)
      ANI     M229  ; 強制運轉模式
      ORB
      AND     M80  ; 主傳動允許運轉
      ANI     M1703  ; 主傳動卡板偵測異常
      ANI     M83  ; 主傳動定位到達
      OUT     Y119  ; 主傳動馬達INV20反轉(往出料)
      ANI     M232  ; 自動模式KP
      ANI     M229  ; 強制運轉模式
      OUT     M111  ; 手動步進一次燈
380   LD      M87  ; 強制往進料方向
      AND     M80  ; 主傳動允許運轉
      OUT     Y118  ; 主傳動運轉往入料
383   LDI     M229  ; 強制運轉模式
      MPS
      ANI     X0  ; 主傳動左定位
      ANI     X1  ; 主傳動右定位
      AND     Y119  ; 主傳動馬達INV20反轉(往出料)
      OUT     T10 K2  ; 主傳動定位脫離偵測延遲
      MPP
      AND     Y119  ; 主傳動馬達INV20反轉(往出料)
      LD      T10  ; 主傳動定位脫離偵測延遲
      OR      M82  ; 主傳動定位脫離KP
      ANB
      OUT     M82  ; 主傳動定位脫離KP
      AND     M1300  ; 主傳動定位到達
      OUT     M83  ; 主傳動定位到達
400   END
END_PROGRAM

PROGRAM 16ETHERN
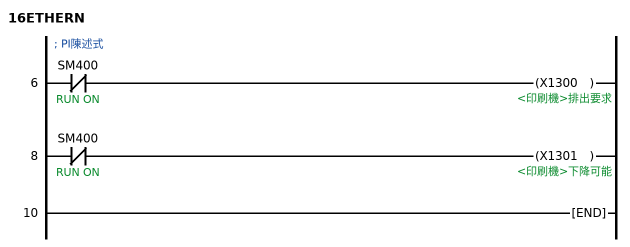
; PI陳述式
6     LDI     SM400  ; RUN ON
      OUT     X1300  ; <印刷機>排出要求
8     LDI     SM400  ; RUN ON
      OUT     X1301  ; <印刷機>下降可能
10    END
END_PROGRAM

PROGRAM 17GBF-20
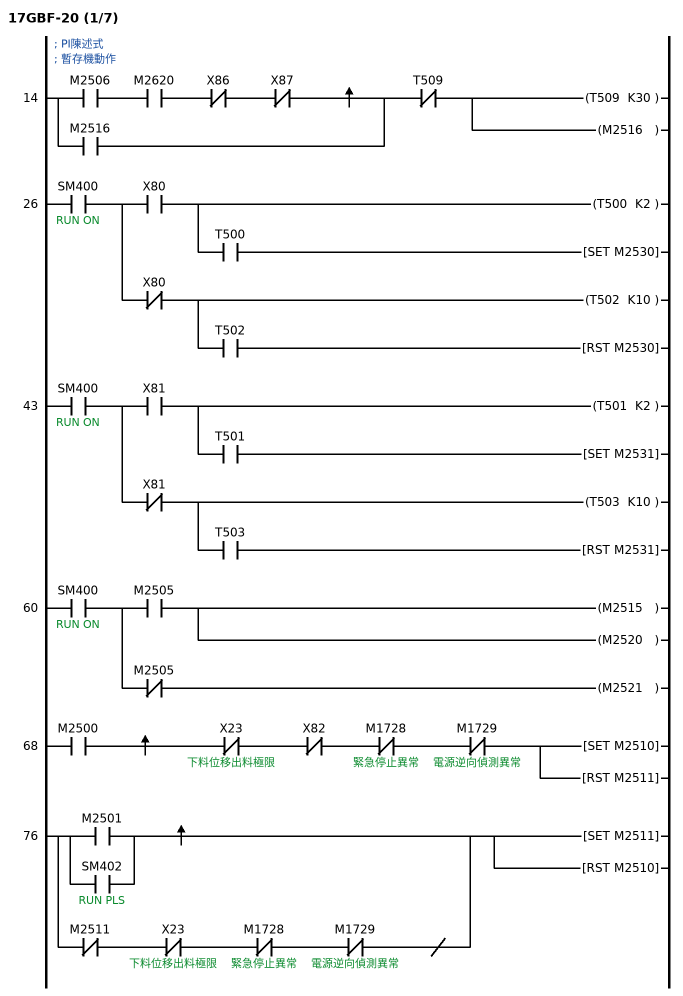
; PI陳述式
; 暫存機動作
14    LD      M2506
      AND     M2620
      ANI     X86
      ANI     X87
      MEP
      OR      M2516
      ANI     T509
      OUT     T509 K30
      OUT     M2516
26    LD      SM400  ; RUN ON
      MPS
      AND     X80
      OUT     T500 K2
      AND     T500
      SET     M2530
      MPP
      ANI     X80
      OUT     T502 K10
      AND     T502
      RST     M2530
43    LD      SM400  ; RUN ON
      MPS
      AND     X81
      OUT     T501 K2
      AND     T501
      SET     M2531
      MPP
      ANI     X81
      OUT     T503 K10
      AND     T503
      RST     M2531
60    LD      SM400  ; RUN ON
      MPS
      AND     M2505
      OUT     M2515
      OUT     M2520
      MPP
      ANI     M2505
      OUT     M2521
68    LD      M2500
      MEP
      ANI     X23  ; 下料位移出料極限
      ANI     X82
      ANI     M1728  ; 緊急停止異常
      ANI     M1729  ; 電源逆向偵測異常
      SET     M2510
      RST     M2511
76    LD      M2501
      OR      SM402  ; RUN PLS
      MEP
      LDI     M2511
      ANI     X23  ; 下料位移出料極限
      ANI     M1728  ; 緊急停止異常
      ANI     M1729  ; 電源逆向偵測異常
      INV
      ORB
      SET     M2511
      RST     M2510
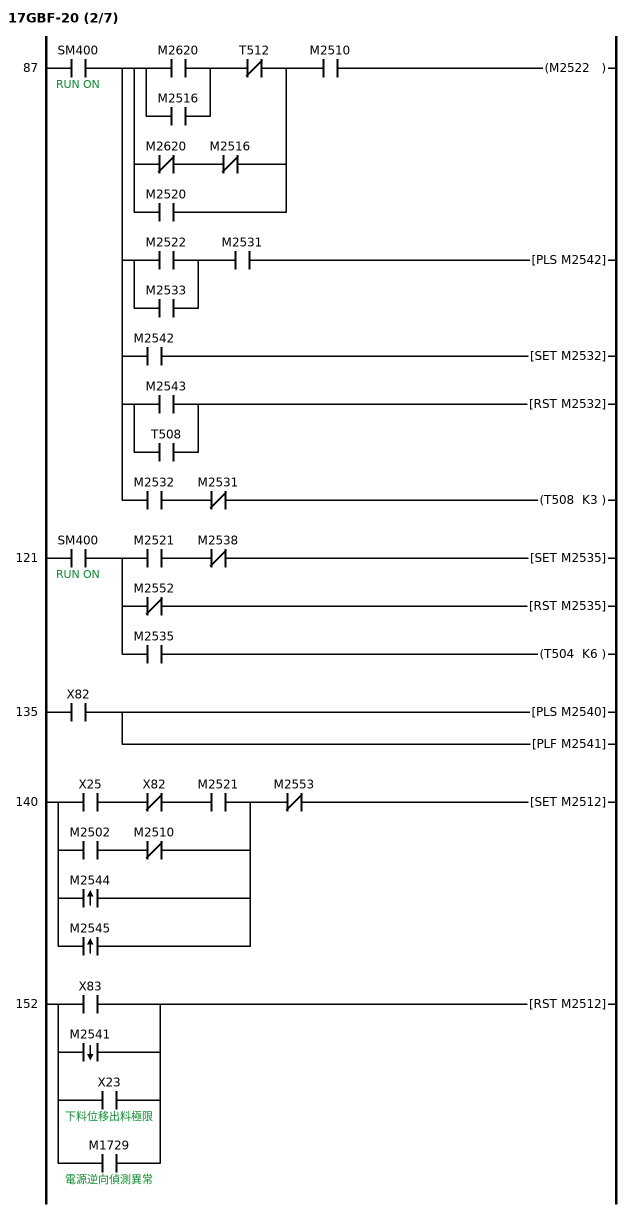
87    LD      SM400  ; RUN ON
      MPS
      LD      M2620
      OR      M2516
      ANI     T512
      LDI     M2620
      ANI     M2516
      ORB
      OR      M2520
      ANB
      AND     M2510
      OUT     M2522
      MRD
      LD      M2522
      OR      M2533
      ANB
      AND     M2531
      PLS     M2542
      MRD
      AND     M2542
      SET     M2532
      MRD
      LD      M2543
      OR      T508
      ANB
      RST     M2532
      MPP
      AND     M2532
      ANI     M2531
      OUT     T508 K3
121   LD      SM400  ; RUN ON
      MPS
      AND     M2521
      ANI     M2538
      SET     M2535
      MRD
      ANI     M2552
      RST     M2535
      MPP
      AND     M2535
      OUT     T504 K6
135   LD      X82
      PLS     M2540
      PLF     M2541
140   LD      X25
      ANI     X82
      AND     M2521
      LD      M2502
      ANI     M2510
      ORB
      ORP     M2544
      ORP     M2545
      ANI     M2553
      SET     M2512
152   LD      X83
      ORF     M2541
      OR      X23  ; 下料位移出料極限
      OR      M1729  ; 電源逆向偵測異常
      RST     M2512
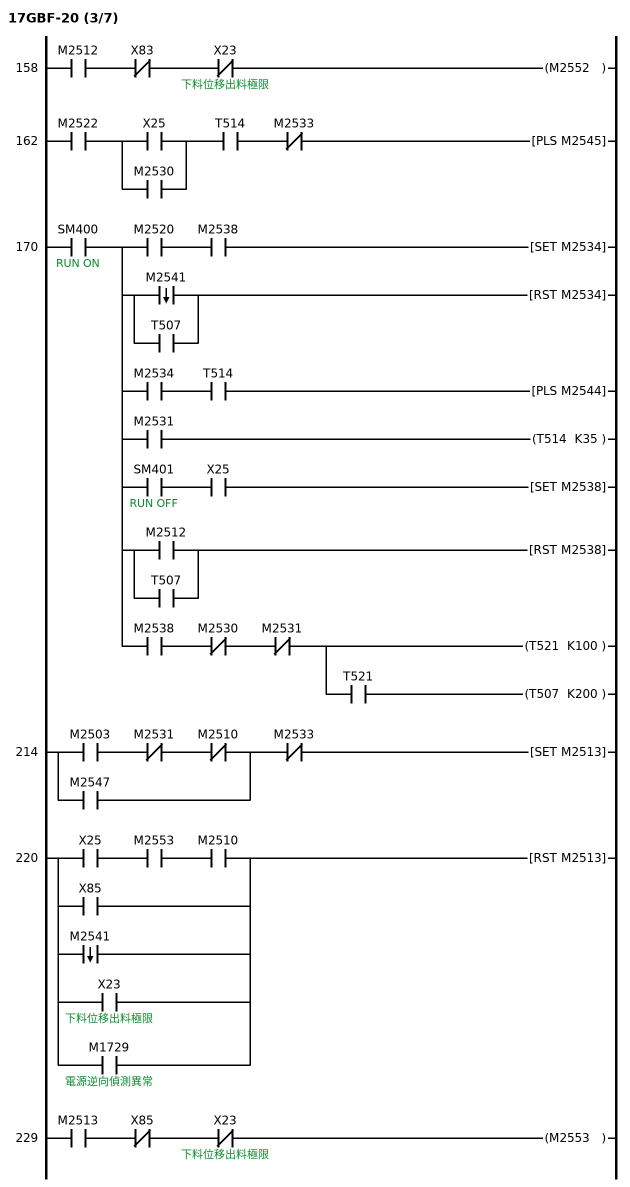
158   LD      M2512
      ANI     X83
      ANI     X23  ; 下料位移出料極限
      OUT     M2552
162   LD      M2522
      LD      X25
      OR      M2530
      ANB
      AND     T514
      ANI     M2533
      PLS     M2545
170   LD      SM400  ; RUN ON
      MPS
      AND     M2520
      AND     M2538
      SET     M2534
      MRD
      LDF     M2541
      OR      T507
      ANB
      RST     M2534
      MRD
      AND     M2534
      AND     T514
      PLS     M2544
      MRD
      AND     M2531
      OUT     T514 K35
      MRD
      AND     SM401  ; RUN OFF
      AND     X25
      SET     M2538
      MRD
      LD      M2512
      OR      T507
      ANB
      RST     M2538
      MPP
      AND     M2538
      ANI     M2530
      ANI     M2531
      OUT     T521 K100
      AND     T521
      OUT     T507 K200
214   LD      M2503
      ANI     M2531
      ANI     M2510
      OR      M2547
      ANI     M2533
      SET     M2513
220   LD      X25
      AND     M2553
      AND     M2510
      OR      X85
      ORF     M2541
      OR      X23  ; 下料位移出料極限
      OR      M1729  ; 電源逆向偵測異常
      RST     M2513
229   LD      M2513
      ANI     X85
      ANI     X23  ; 下料位移出料極限
      OUT     M2553
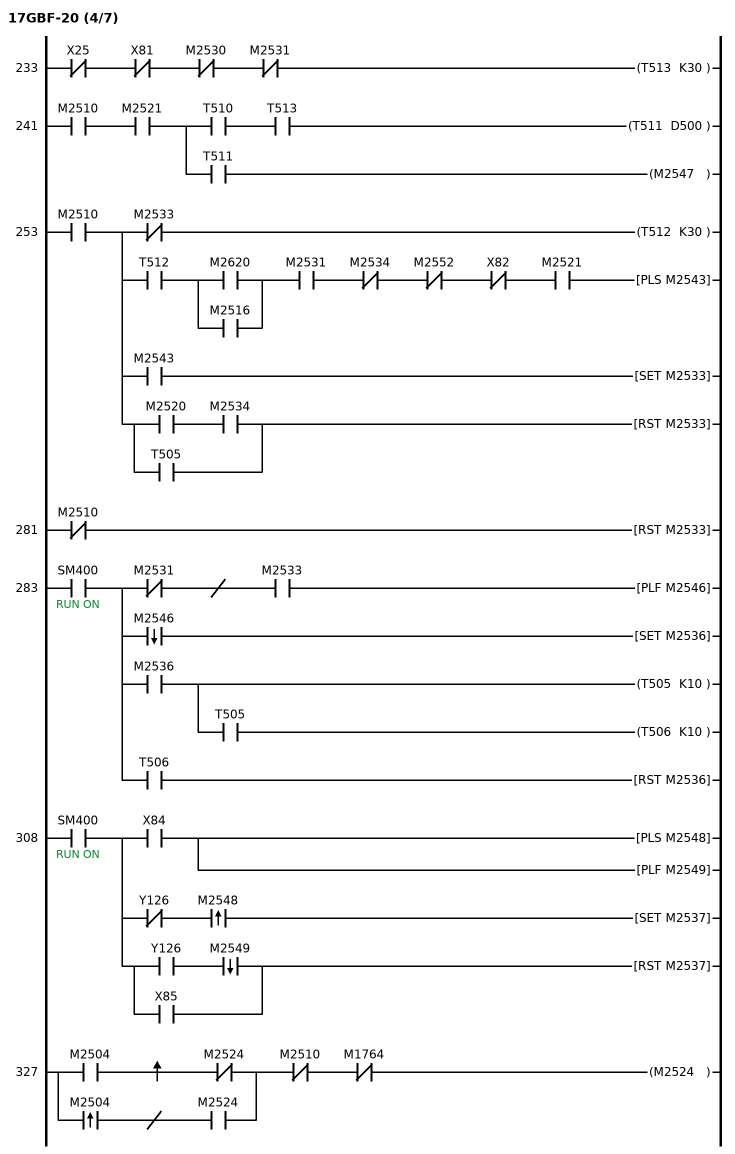
233   LDI     X25
      ANI     X81
      ANI     M2530
      ANI     M2531
      OUT     T513 K30
241   LD      M2510
      AND     M2521
      MPS
      AND     T510
      AND     T513
      OUT     T511 D500
      MPP
      AND     T511
      OUT     M2547
253   LD      M2510
      MPS
      ANI     M2533
      OUT     T512 K30
      MRD
      AND     T512
      LD      M2620
      OR      M2516
      ANB
      AND     M2531
      ANI     M2534
      ANI     M2552
      ANI     X82
      AND     M2521
      PLS     M2543
      MRD
      AND     M2543
      SET     M2533
      MPP
      LD      M2520
      AND     M2534
      OR      T505
      ANB
      RST     M2533
281   LDI     M2510
      RST     M2533
283   LD      SM400  ; RUN ON
      MPS
      ANI     M2531
      INV
      AND     M2533
      PLF     M2546
      MRD
      ANDF    M2546
      SET     M2536
      MRD
      AND     M2536
      OUT     T505 K10
      AND     T505
      OUT     T506 K10
      MPP
      AND     T506
      RST     M2536
308   LD      SM400  ; RUN ON
      MPS
      AND     X84
      PLS     M2548
      PLF     M2549
      MRD
      ANI     Y126
      ANDP    M2548
      SET     M2537
      MPP
      LD      Y126
      ANDF    M2549
      OR      X85
      ANB
      RST     M2537
327   LD      M2504
      MEP
      ANI     M2524
      LDP     M2504
      INV
      AND     M2524
      ORB
      ANI     M2510
      ANI     M1764
      OUT     M2524
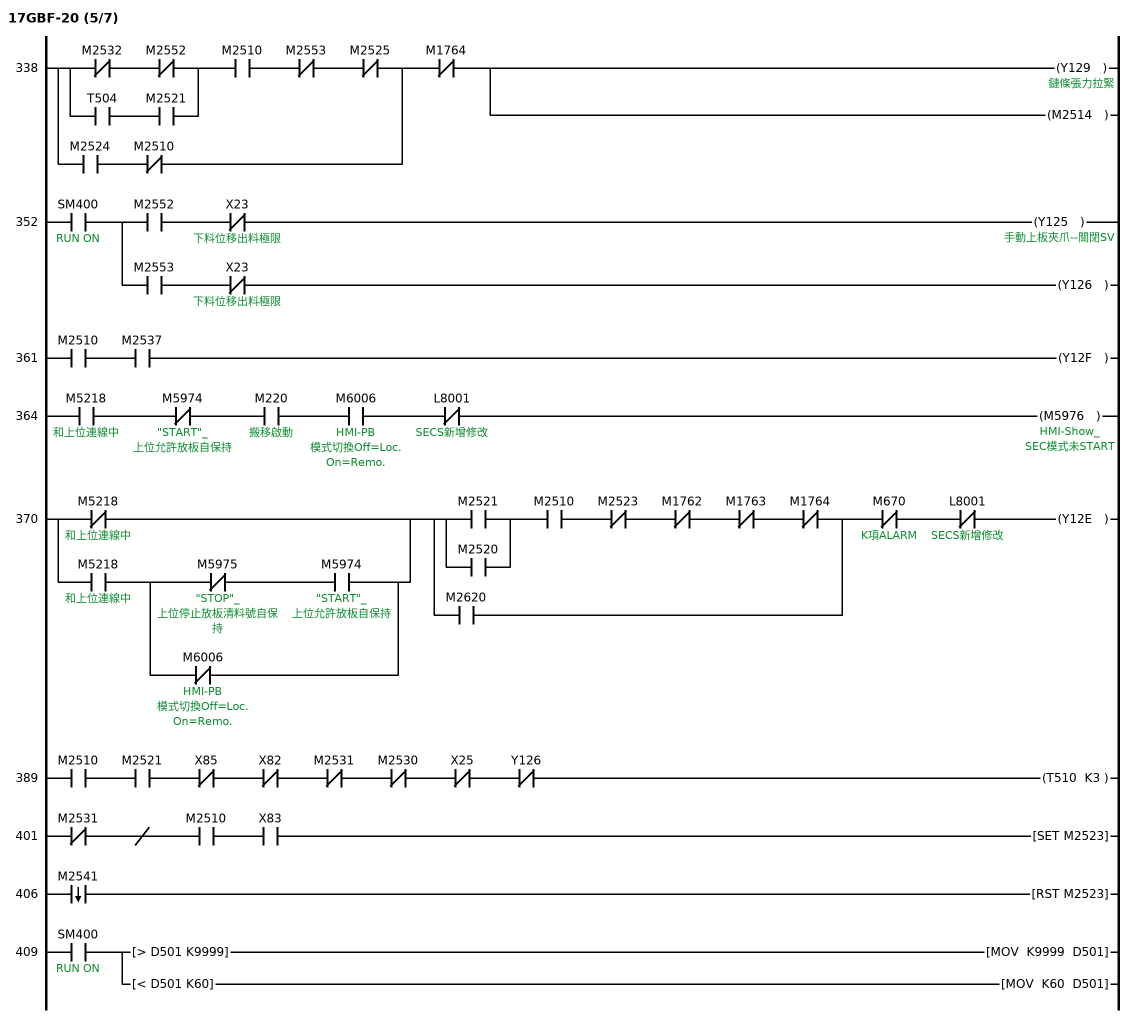
338   LDI     M2532
      ANI     M2552
      LD      T504
      AND     M2521
      ORB
      AND     M2510
      ANI     M2553
      ANI     M2525
      LD      M2524
      ANI     M2510
      ORB
      ANI     M1764
      OUT     Y129  ; 鏈條張力拉緊
      OUT     M2514
352   LD      SM400  ; RUN ON
      MPS
      AND     M2552
      ANI     X23  ; 下料位移出料極限
      OUT     Y125  ; 手動上板夾爪--關閉SV
      MPP
      AND     M2553
      ANI     X23  ; 下料位移出料極限
      OUT     Y126
361   LD      M2510
      AND     M2537
      OUT     Y12F
364   LD      M5218  ; 和上位連線中
      ANI     M5974  ; "START"_上位允許放板自保持
      AND     M220  ; 搬移啟動
      AND     M6006  ; HMI-PB  模式切換Off=Loc.On=Remo.
      ANI     L8001  ; SECS新增修改
      OUT     M5976  ; HMI-Show_SEC模式未START
370   LDI     M5218  ; 和上位連線中
      LD      M5218  ; 和上位連線中
      LDI     M5975  ; "STOP"_ 上位停止放板清料號自保持
      AND     M5974  ; "START"_上位允許放板自保持
      ORI     M6006  ; HMI-PB  模式切換Off=Loc.On=Remo.
      ANB
      ORB
      LD      M2521
      OR      M2520
      AND     M2510
      ANI     M2523
      ANI     M1762
      ANI     M1763
      ANI     M1764
      OR      M2620
      ANB
      ANI     M670  ; K項ALARM
      ANI     L8001  ; SECS新增修改
      OUT     Y12E
389   LD      M2510
      AND     M2521
      ANI     X85
      ANI     X82
      ANI     M2531
      ANI     M2530
      ANI     X25
      ANI     Y126
      OUT     T510 K3
401   LDI     M2531
      INV
      AND     M2510
      AND     X83
      SET     M2523
406   LDF     M2541
      RST     M2523
409   LD      SM400  ; RUN ON
      MPS
      AND>    D501 K9999
      MOV     K9999 D501
      MPP
      AND<    D501 K60
      MOV     K60 D501
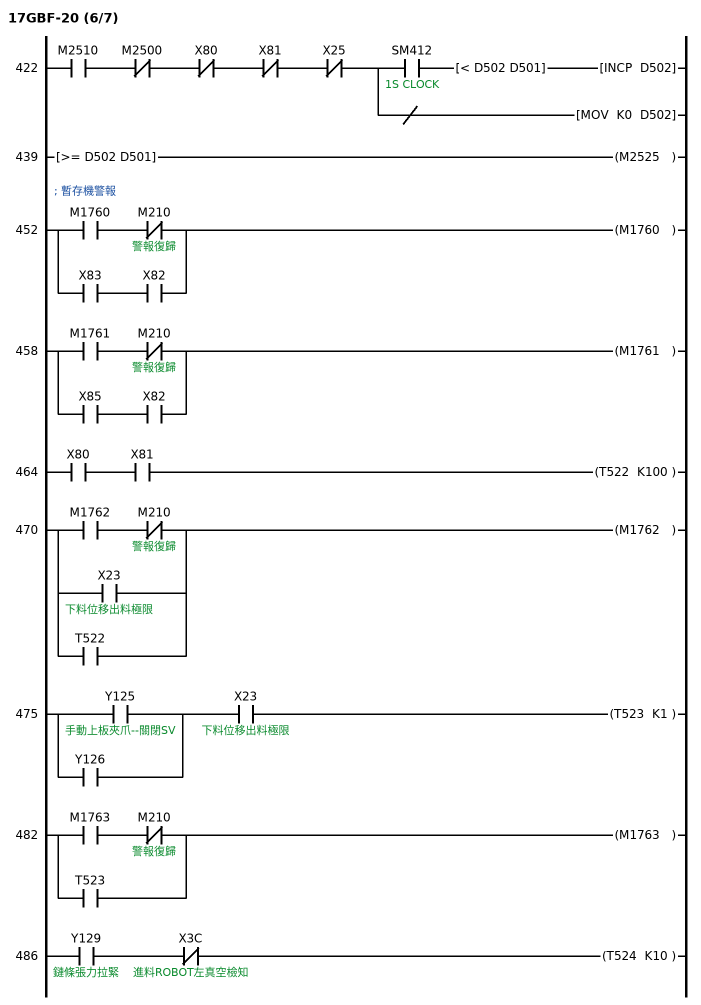
422   LD      M2510
      ANI     M2500
      ANI     X80
      ANI     X81
      ANI     X25
      MPS
      AND     SM412  ; 1S CLOCK
      AND<    D502 D501
      INCP    D502
      MPP
      INV
      MOV     K0 D502
439   LD>=    D502 D501
      OUT     M2525
; 暫存機警報
452   LD      M1760
      ANI     M210  ; 警報復歸
      LD      X83
      AND     X82
      ORB
      OUT     M1760
458   LD      M1761
      ANI     M210  ; 警報復歸
      LD      X85
      AND     X82
      ORB
      OUT     M1761
464   LD      X80
      AND     X81
      OUT     T522 K100
470   LD      M1762
      ANI     M210  ; 警報復歸
      OR      X23  ; 下料位移出料極限
      OR      T522
      OUT     M1762
475   LD      Y125  ; 手動上板夾爪--關閉SV
      OR      Y126
      AND     X23  ; 下料位移出料極限
      OUT     T523 K1
482   LD      M1763
      ANI     M210  ; 警報復歸
      OR      T523
      OUT     M1763
486   LD      Y129  ; 鏈條張力拉緊
      ANI     X3C  ; 進料ROBOT左真空檢知
      OUT     T524 K10
